// TIA Portal V21 export
VAR_GLOBAL   // PLC tag table "K_TipoAccoppiamentoUscitePid"
END_VAR
VAR_GLOBAL CONSTANT   // user constants
   K_TipoAccoppiamentoUscitePid_Uguali : Int := 0;   // Le due utenze in uscita ricevono il 0-100% Del PID allo stesso modo
   K_TipoAccoppiamentoUscitePid_PosNeg : Int := 1;   // L'uscita viene scalata da 0-50PID / 0-100%CmdNeg | 50-100PID / 0-100%CmdPos
END_VAR
